FUNCTION_BLOCK T_RoboConnect_GetToolDigitalOutput_IncorrectIndexFails EXTENDS T_UnitTestBase
VAR
  robot : I_RoboConnect;
  targetDO : UINT;
  myTestState, prevState :
    (INIT,
    ARRANGE,
    ACT,
    ASSERT) := INIT;
  expected : BOOL;
  actual : BOOL := TRUE;
  counter : UINT;
  returnedTask : I_Task;
  resultTask : I_BoolResultTask;
END_VAR

CASE myTestState OF
  INIT:
    StateChanged();
    myTestState := ARRANGE;

  ARRANGE:
    IF StateChanged() THEN
      expected := FALSE;
      myTestState := ACT;
    END_IF

  ACT:
    actual := robot.GetToolDigitalOutput(targetDO, task => resultTask);
    myTestState := ASSERT;

  ASSERT:
    assertion.AssertEquals_BOOL(expected, actual, 'robot.GetToolDigitalOutput(targetDO, task => returnedTask)');
    TestFinished();
    myTestState := INIT;

END_CASE

METHOD FB_init : BOOL
VAR_INPUT
  bInitRetains : BOOL; // if TRUE, the retain variables are initialized (warm start / cold start)
  bInCopyCode : BOOL; // if TRUE, the instance afterwards gets moved into the copy code (online change)
  TestSuite : tcl_SimpleUnitTestLibrary.I_TestSuite;
  robot : I_TcRobot;
  targetDo : UINT;
END_VAR
THIS^.robot := robot;
THIS^.targetDo := targetDo;
END_METHOD

METHOD PRIVATE StateChanged : BOOL
IF  myTestState = prevState THEN
  RETURN;
END_IF

prevState := myTestState;
StateChanged := TRUE;
END_METHOD

METHOD WaitForCycles : BOOL
VAR_INPUT
  maxCount : UINT;
END_VAR
counter := counter + 1;

IF counter = maxCount THEN
  counter := 0;
  WaitForCycles := TRUE;
END_IF
END_METHOD

END_FUNCTION_BLOCK

(* stored: Version 1.1.0.1
   POU T_TcRobot_GetToolDigitalOutput_IncorrectIndexFails: Id {8a67c7da-1615-4525-a5f4-d3c2c793dc88}, SpecialFunc None
   Method FB_init: Id {2dda81c4-70e6-4cf5-8fd7-94fb1d9df12d}
   Method StateChanged: Id {3fbf2039-8ea8-49b6-bb36-4f03ca8b0dcd}
   Method WaitForCycles: Id {f00b7ddb-790b-4e83-9fcb-7d49c3775a5e} *)
